PROGRAM P_AUTOMATION
VAR
END_VAR

END_PROGRAM

(* stored: Version 1.1.0.1, ProductVersion 3.1.4024.10
   POU P_AUTOMATION: Id {533f5014-8755-47f8-a5a5-ad530ab45145}, SpecialFunc None *)
